// TIA Portal V17 export
// export: Created 2022-05-07T16:38:47.4456513Z, ExportSetting WithDefaults, DisplayName Totally Integrated Automation Portal, DisplayVersion V17 Update 3, DisplayName TIA Portal Openness, DisplayVersion V17 Update 3, DisplayName TIA Portal Version Control Interface, DisplayVersion V17, DisplayName TIA Portal Test Suite Advanced, DisplayVersion V17 Update 1, DisplayName SINAMICS Startdrive Advanced, DisplayVersion V17 Update2, DisplayName SINAMICS Startdrive G130, G150, S120, S150, SINAMICS MV, S210, DisplayVersion V17 Update2, DisplayName SINAMICS Startdrive G110M, G120, G120C, G120D, G120P, G115D, DisplayVersion V17 Update2, DisplayName STEP 7 Professional, DisplayVersion V17 Update 3, DisplayName STEP 7 Safety, DisplayVersion V17, DisplayName WinCC UA Professional, DisplayVersion V17 Update 3
FUNCTION_BLOCK "FB_STATI_MACCHINA"   // FB2, LAD
{ S7_Optimized_Access := 'TRUE' }
VERSION : 0.1
// stored: AutoNumber true, IsIECCheckEnabled false, IsRetainMemResEnabled false, MemoryReserve 100, SetENOAutomatically false, UDAEnableTagReadback false
   VAR
      TAux { S7_SetPoint := 'True'} : TON_TIME;
      TResetAlla { S7_SetPoint := 'True'} : TON_TIME;
   END_VAR
BEGIN

REGION Network 1: AUX OK
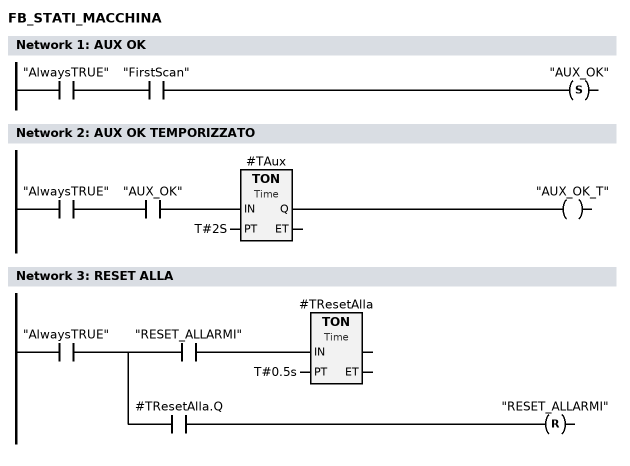
   RUNG wire#powerrail
      Contact( "AlwaysTRUE" )
      Contact( "FirstScan" )
      S_Coil( "AUX_OK" )
   END_RUNG
   // the same network as SCL:
   IF "AlwaysTRUE" AND "FirstScan" THEN "AUX_OK" := TRUE; END_IF;
END_REGION

REGION Network 2: AUX OK TEMPORIZZATO
   RUNG wire#powerrail
      Contact( "AlwaysTRUE" )
      Contact( "AUX_OK" )
      { S7_Templates := "time_type := Time" } #TAux.TON(pt := T#2S, et =>)
      Coil( "AUX_OK_T" )
   END_RUNG
   // the same network as SCL:
   #TAux(IN := "AlwaysTRUE" AND "AUX_OK", PT := T#2S);   // TON
   "AUX_OK_T" := #TAux.Q;
END_REGION

REGION Network 3: RESET ALLA
   RUNG wire#powerrail
      Contact( "AlwaysTRUE" )
      wire#w1
      Contact( "RESET_ALLARMI" )
      { S7_Templates := "time_type := Time" } #TResetAlla.TON(pt := T#0.5s, et =>)
   END_RUNG
   RUNG wire#w1
      Contact( #TResetAlla.Q )
      R_Coil( "RESET_ALLARMI" )
   END_RUNG
   // the same network as SCL:
   #TResetAlla(IN := "AlwaysTRUE" AND "RESET_ALLARMI", PT := T#0.5s);   // TON
   IF "AlwaysTRUE" AND #TResetAlla.Q THEN "RESET_ALLARMI" := FALSE; END_IF;
END_REGION

REGION Network 4 (SCL): MAN/AUTO

   "MANUALE" := NOT "AUTOMATICO";
END_REGION
END_FUNCTION_BLOCK
